// TIA Portal V17 export
// export: Created 2024-09-02T12:50:35.676165Z, ExportSetting WithDefaults, DisplayName Totally Integrated Automation Portal, DisplayVersion V17, DisplayName TIA Portal Openness, DisplayVersion V17, DisplayName TIA Portal Version Control Interface, DisplayVersion V17, DisplayName STEP 7 Professional, DisplayVersion V17, DisplayName STEP 7 Safety, DisplayVersion V17, DisplayName WinCC Professional, DisplayVersion V17
TYPE "TypeMobyAnbauteile_1"
// stored: IsFailsafeCompliant false
   STRUCT
      Alternativ_1 { S7_SetPoint := 'True'} : "TypeMobyAnbauteil_1";   // Scancode Alternativ 1 Bauteil Soll / Scancode Alternative 1 Component Target
      Alternativ_2 { S7_SetPoint := 'True'} : "TypeMobyAnbauteil_1";   // Scancode Alternativ 2 Bauteil Soll / Scancode Alternative 2 Component Target
      Alternativ_3 { S7_SetPoint := 'True'} : "TypeMobyAnbauteil_1";   // Scancode Alternativ 3 Bauteil Soll / Scancode Alternative 3 Component Target
      Alternativ_4 { S7_SetPoint := 'True'} : "TypeMobyAnbauteil_1";   // Scancode Alternativ 4 Bauteil Soll / Scancode Alternative 4 Component Target
      Alternativ_5 { S7_SetPoint := 'True'} : "TypeMobyAnbauteil_1";   // Scancode Alternativ 5 Bauteil Soll / Scancode Alternative 5 Component Target
   END_STRUCT;
END_TYPE
